(* Schneider Machine Expert - Basic project water_pump_and_water_level, file version 2.7.0.0 *)
(* ProjectInformations: Name=New project *)

HARDWARE
  Cpu 0: TM221M16R/G
  EthernetConfiguration: NetworkName=M221, IpAllocationMode=FixedAddress, IpAddress=0.0.0.0, SubnetMask=0.0.0.0
  SerialLineConfiguration: Baud=Baud19200, Parity=ParityEven, DataBits=DataBits8, StopBits=StopBits1, PhysicalMedium=PhysicalMediumRs485, TransmissionMode=TransmissionModeModbusRtu, SlaveId=1, Addressing=SlaveAddressing
  MastTask: UsePeriodScanMode=false, PeriodScan=100
  FastTask: Period=255
  CpuBehavior: StartingMode=StartAsPreviousState, AutoSaveRamOnEeprom=true, WatchdogPeriod=250

SYMBOLS  (address, symbol, comment, settings)
  %M0       IS_START
  %I0.0     STARTING
  %I0.1     STOP
  %I0.2     LLS
  %I0.3     HLS
  %Q0.0     PUMP_IT

POU New POU
  (* SectionNumber=1 *)

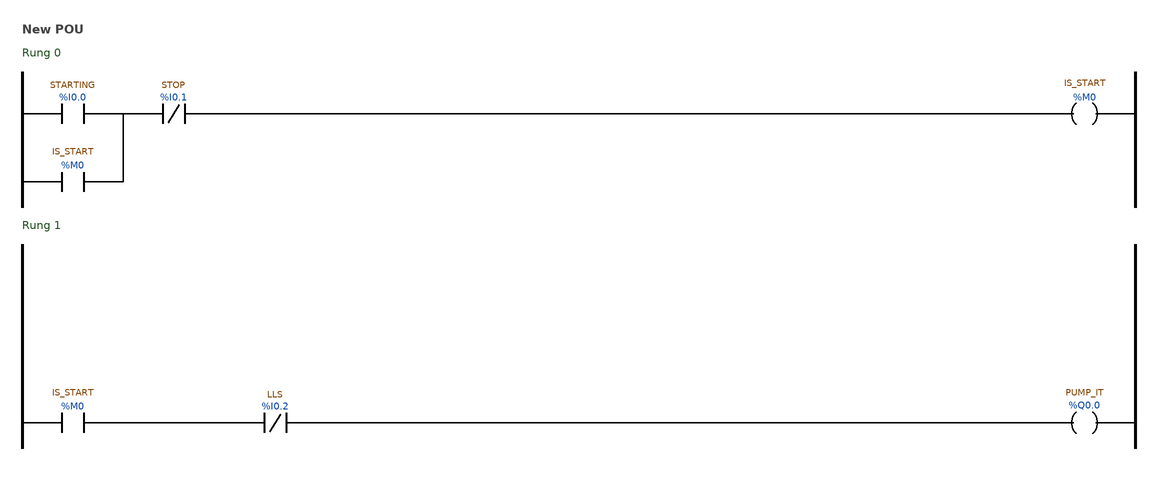

// Rung 0
  LD %I0.0                (* STARTING *)
  OR %M0                  (* IS_START *)
  ANDN %I0.1              (* STOP *)
  ST %M0                  (* IS_START *)
  // as ST:
  //   IS_START := (STARTING OR IS_START) AND NOT STOP;

// Rung 1
  LD %M0                  (* IS_START *)
  ANDN %I0.2              (* LLS *)
  ST %Q0.0                (* PUMP_IT *)
  // as ST:
  //   PUMP_IT := IS_START AND NOT LLS;
